TYPE SL_INSTRUCTIONS :
STRUCT
	Line : STRING(255);
END_STRUCT
END_TYPE

(* stored: Version 1.1.0.1, ProductVersion 3.1.4024.10
   DUT SL_INSTRUCTIONS: Id {db56f2e0-8d60-4cef-9beb-a82349e60923} *)
